Fanuc KAREL source: KA00181.KL

PROGRAM KA00181
%NOLOCKGROUP
VAR
  SRC: ARRAY[4] OF BYTE
  DST: ARRAY[4] OF INTEGER
BEGIN
  DST = SRC
END KA00181
